Staubli VAL3: compareStr.pgx

public program compareStr(string& x_sInput[], string x_sCompareTo, bool& x_bResult[])
  local num l_nLength
  local num l_nElement
begin

  l_nLength = size(x_sInput)
  x_bResult[0] = false
  resize(x_bResult,1,l_nLength)

  for l_nElement = 0 to l_nLength-1
    if x_sInput[l_nElement] == x_sCompareTo
      x_bResult[l_nElement] = true
    else
      x_bResult[l_nElement] = false
    endIf
  endFor
end
